FUNCTION_BLOCK FB_WriteCoE

VAR_INPUT
	sNetId			: T_AmsNetId;
	nSlaveAddr 		: UINT;
	nIndex			: WORD;
	nIndexOffset	: BYTE;
	nParameter		: INT;
END_VAR

VAR_OUTPUT
	bDoneWriting	: BOOL;
	bError			: BOOL;
END_VAR

VAR
	bExecute		: BOOL;
	fbCoeWrite		: FB_EcCoEsDoWrite;
	eCoEWriteState	: (INIT, TRIGGER, WRITE, DONE);
END_VAR

CASE eCoEWriteState OF
	
	INIT:
		bDoneWriting := FALSE;
		bExecute := FALSE;
		eCoEWriteState := TRIGGER;
		
	TRIGGER:
		bExecute := TRUE;
		eCoEWriteState := WRITE;
		
	WRITE:
		fbCoeWrite(
			sNetId:=sNetId, 
			nSlaveAddr:=nSlaveAddr, 
			nSubIndex:=nIndexOffset, 
			nIndex:=nIndex, 
			pSrcBuf:=ADR(nParameter), 
			cbBufLen:=SIZEOF(nParameter), 
			bExecute:=bExecute);
			
		bExecute := NOT bExecute;
		
		IF NOT fbCoeWrite.bBusy THEN
			eCoeWriteState := DONE;
		END_IF
	
	DONE:
		IF fbCoeWrite.bError THEN
			bError := TRUE;
		ELSE
			bError := FALSE;
		END_IF
		bDoneWriting := TRUE;
		eCoEWriteState := INIT;
		
END_CASE

END_FUNCTION_BLOCK

(* stored: Version 1.1.0.1, ProductVersion 3.1.4024.9
   POU FB_WriteCoE: Id {09573ff6-d8b7-42fc-b85e-49366cf46ffa}, SpecialFunc None *)
